{attribute 'enable_dynamic_creation'}
FUNCTION_BLOCK FutureGripperControl EXTENDS FB_AbstructFuture
VAR_INPUT
END_VAR
VAR_OUTPUT
END_VAR
VAR
	_gripper_close_output : REFERENCE TO BOOL;
	_gripper_open_output : REFERENCE TO BOOL;
	_gripper_closed_sensor : REFERENCE TO BOOL;
	_gripper_open_sensor : REFERENCE TO BOOL;
	_command : BOOL; // TRUE = Close, FALSE = Open
	_timeout_timer : TON;
	_timeout_value : TIME := T#5S;
	_error_id : UDINT;
	_exec_state : UDINT;
END_VAR

METHOD execute : BOOL
CASE _exec_state OF
	0: // Start gripper operation
		_timeout_timer(IN := FALSE);
		
		IF _command THEN // Close gripper
			_gripper_close_output := TRUE;
			_gripper_open_output := FALSE;
		ELSE // Open gripper
			_gripper_close_output := FALSE;
			_gripper_open_output := TRUE;
		END_IF
		
		_exec_state := 1;
		
	1: // Wait for gripper to reach position
		_timeout_timer(IN := TRUE, PT := _timeout_value);
		
		IF _command THEN // Closing - wait for closed sensor
			IF _gripper_closed_sensor THEN
				_error_id := 0;
				execute := TRUE;
			ELSIF _timeout_timer.Q THEN
				_error_id := 16#8001; // Gripper close timeout error
				execute := TRUE;
			END_IF
		ELSE // Opening - wait for open sensor
			IF _gripper_open_sensor THEN
				_error_id := 0;
				execute := TRUE;
			ELSIF _timeout_timer.Q THEN
				_error_id := 16#8002; // Gripper open timeout error
				execute := TRUE;
			END_IF
		END_IF
END_CASE

_timeout_timer();
END_METHOD

METHOD init : BOOL
_exec_state := 0;
_error_id := 0;
_timeout_timer(IN := FALSE);
init := TRUE;
END_METHOD

PROPERTY nErrorID : UDINT
GET
nErrorID := _error_id;
END_GET
SET
END_SET
END_PROPERTY

METHOD set_parameters : BOOL
VAR_INPUT
	gripper_close_output : REFERENCE TO BOOL;
	gripper_open_output : REFERENCE TO BOOL;
	gripper_closed_sensor : REFERENCE TO BOOL;
	gripper_open_sensor : REFERENCE TO BOOL;
	command : BOOL; // TRUE = Close, FALSE = Open
	timeout : TIME := T#5S;
END_VAR
_gripper_close_output REF= gripper_close_output;
_gripper_open_output REF= gripper_open_output;
_gripper_closed_sensor REF= gripper_closed_sensor;
_gripper_open_sensor REF= gripper_open_sensor;
_command := command;
_timeout_value := timeout;
set_parameters := TRUE;
END_METHOD

END_FUNCTION_BLOCK

(* stored: Version 1.1.0.1, ProductVersion 3.1.4024.12
   POU FutureGripperControl: Id {12345678-1234-1234-1234-123456789abc}, SpecialFunc None
   Method execute: Id {12345678-1234-1234-1234-123456789def}
   Method init: Id {12345678-1234-1234-1234-123456789fed}
   Property nErrorID: Id {12345678-1234-1234-1234-123456789cba}
   Get Get: Id {12345678-1234-1234-1234-123456789dfe}
   Set Set: Id {12345678-1234-1234-1234-123456789ced}
   Method set_parameters: Id {12345678-1234-1234-1234-123456789bcd} *)
